// TIA Portal V20 export
FUNCTION_BLOCK "1500Diag82"   // FB82, SCL
{ S7_Optimized_Access := 'TRUE' }
VERSION : 1.1
// stored: MemoryReserve 100, SetENOAutomatically false
   VAR_INPUT
      fId : HW_IO;   // HW-Id of the component from which interrupts are to be received
   END_VAR
   VAR_OUTPUT
      new : Bool;   // A new interrupt was received.
      status : DWord;   // Function result/error message
      id : HW_IO;   // HW-Id of the component (module) from which an interrupt was received
      len : UInt;   // Length of the received interrupt information
      areaLenError : Bool;   // Area length error
   END_VAR
   VAR_IN_OUT
      diag : "typeDiag";   // diagnostics data
   END_VAR
   VAR
      statTinfo { S7_SetPoint := 'True'} : TI_DiagnosticInterrupt;   // Destination area for OB start and management information
      statAinfo { S7_SetPoint := 'True'} : "typeAiPnOrCentral";   // Destination area for header information and additional interrupt information
      statErrorType : USInt;   // Type of error
      statChannelType : USInt;   // Type of channel
      instRalrm { S7_SetPoint := 'True'} : RALRM;   // Instance of RALRM
   END_VAR
   VAR_TEMP
      tempIndex : SInt;
      tempUsint : USInt;
      tempInfo : SInt;
      tempMax : SInt;
      tempReal : Real;
   END_VAR
BEGIN
   //=============================================================================
   // SIEMENS AG
   // (c)Copyright 2017
   //-----------------------------------------------------------------------------
   // Library:       -
   // Tested with:   CPU 1512C-1 PN FW V2.0
   // Engineering:   TIA Portal V14 Update1
   // Restrictions:  call in Diagnostic Error Interrupt OB 82
   // Requirements:  SIMATIC S7-1500 CPU
   // Functionality: Channel diagnostics (PROFINET IO or central I/O)
   //-----------------------------------------------------------------------------
   // Change log table:
   // Version  Date        Expert in charge                 Changes applied
   // 02.00.00 12.01.2017  SIMATIC Industry Online Support  New function: ModuleDiag
   //                                                       & multiple-channelDiag
   //=============================================================================

   // call RALRM in MODE 2 with given F_ID
   #instRalrm(MODE := 2,
              F_ID := #fId,
              NEW => #new,
              STATUS => #status,
              ID => #id,
              LEN => #len,
              TINFO := #statTinfo,
              AINFO := #statAinfo);

   IF (#id = #fId) // some infos will be read every call of OB82
     AND (#statAinfo.addInfo.formatIdentifier = W#16#8000) THEN // W#16#8000: Channel diagnostics 

     #diag.multiError := #statTinfo.MultiError; // =TRUE, if there is more than one error.
     #diag.slotNumber := #statAinfo.header.slotNumber; // Slot number of the component triggering the interrupt
     #diag.submoduleSlotNumber := #statAinfo.header.submoduleSlotNumber; // Submodule slot number of the component triggering the interrupt 
     #tempReal := UINT_TO_REAL(#statAinfo.header.blockLength - 24) / 6; // calculate numbers of multiple-channelDiag
     #tempMax := REAL_TO_SINT(#tempReal) - 1; // calculate upper limit for FOR loop

     FOR #tempInfo := 0 TO #tempMax DO // FOR loop for multiple-channelDiag
       #tempUsint := SHL(IN := #statAinfo.addInfo.diag[#tempInfo].channelErrorType, N := 3); // calculate Type of error
       #statErrorType := SHR(IN := #tempUsint, N := 6); // 1: Incoming error; 2: Outgoing error

       #statChannelType := SHR(IN := #statAinfo.addInfo.diag[#tempInfo].channelErrorType, N := 5); // calculate Type of channel
       // 1: Input channel; 2: Output channel
       //=============================================================================
         IF (#statErrorType = 1) THEN // 1: Incoming error
         //-----------------------------------------------------------------------------      
         IF (#statChannelType = 1) THEN // 1: Input channel

           IF #statAinfo.addInfo.diag[#tempInfo].channelNumber = -32768 THEN // identify module with module diagnostics only
             #diag.moduleDiagOnly := TRUE;
             "ModuleDiag"(errorCode := #statAinfo.addInfo.diag[#tempInfo].errorCode,
                          value := TRUE,
                          diag := #diag.input.module,
                          errorCounter := #diag.errorCounter);
           ELSE
             #diag.moduleDiagOnly := FALSE;

             IF ((#statAinfo.addInfo.diag[#tempInfo].channelNumber >= 0) AND // check array limits (lower limit)
               (#statAinfo.addInfo.diag[#tempInfo].channelNumber <= #diag.input.channel.chMax)) THEN // check array limits (upper limit)
               #diag.input.channel.ch[#statAinfo.addInfo.diag[#tempInfo].channelNumber].error := TRUE; // Set error
               #diag.input.channel.ch[#statAinfo.addInfo.diag[#tempInfo].channelNumber].errorCode := #statAinfo.addInfo.diag[#tempInfo].errorCode; // copy error code
               #diag.errorCounter := #diag.errorCounter + 1; // increment error counter
               #diag.input.channel.areaLenError := FALSE; // Reset area length error
             ELSE
               #diag.input.channel.areaLenError := TRUE; // Set area length error
             END_IF;
           END_IF;
           //-----------------------------------------------------------------------------   
         ELSIF (#statChannelType = 2) THEN // 2: Output channel

           IF #statAinfo.addInfo.diag[#tempInfo].channelNumber = -32768 THEN // identify module with module diagnostics only
             #diag.moduleDiagOnly := TRUE;
             "ModuleDiag"(errorCode := #statAinfo.addInfo.diag[#tempInfo].errorCode,
                          value := TRUE,
                          diag := #diag.output.module,
                          errorCounter := #diag.errorCounter);
           ELSE
             #diag.moduleDiagOnly := FALSE;

             IF ((#statAinfo.addInfo.diag[#tempInfo].channelNumber >= 0) AND // check array limits (lower limit)
               (#statAinfo.addInfo.diag[#tempInfo].channelNumber <= #diag.output.channel.chMax)) THEN // check array limits (upper limit)
               #diag.output.channel.ch[#statAinfo.addInfo.diag[#tempInfo].channelNumber].error := TRUE; // Set error
               #diag.output.channel.ch[#statAinfo.addInfo.diag[#tempInfo].channelNumber].errorCode := #statAinfo.addInfo.diag[#tempInfo].errorCode; // copy error code
               #diag.errorCounter := #diag.errorCounter + 1; // increment error counter
               #diag.output.channel.areaLenError := FALSE; // Reset area length error
             ELSE
               #diag.output.channel.areaLenError := TRUE; // Set area length error
             END_IF;
           END_IF;
           //-----------------------------------------------------------------------------  
         ELSIF (#statChannelType = 3) THEN // 3: Input/output channel

           IF #statAinfo.addInfo.diag[#tempInfo].channelNumber = -32768 THEN // identify module with module diagnostics only
             #diag.moduleDiagOnly := TRUE;
             "ModuleDiag"(errorCode := #statAinfo.addInfo.diag[#tempInfo].errorCode,
                          value := TRUE,
                          diag := #diag.inOut.module,
                          errorCounter := #diag.errorCounter);
           ELSE
             #diag.moduleDiagOnly := FALSE;

             IF ((#statAinfo.addInfo.diag[#tempInfo].channelNumber >= 0) AND // check array limits (lower limit)
               (#statAinfo.addInfo.diag[#tempInfo].channelNumber <= #diag.inOut.channel.chMax)) THEN // check array limits (upper limit)
               #diag.inOut.channel.ch[#statAinfo.addInfo.diag[#tempInfo].channelNumber].error := TRUE; // Set error
               #diag.inOut.channel.ch[#statAinfo.addInfo.diag[#tempInfo].channelNumber].errorCode := #statAinfo.addInfo.diag[#tempInfo].errorCode; // copy error code
               #diag.errorCounter := #diag.errorCounter + 1; // increment error counter
               #diag.inOut.channel.areaLenError := FALSE; // Reset area length error
             ELSE
               #diag.inOut.channel.areaLenError := TRUE; // Set area length error
             END_IF;
           END_IF;
         END_IF;
         //=============================================================================  
       ELSIF (#statErrorType >= 2) THEN // 2: Outgoing error; 3: Outgoing error, other errors present
         //-----------------------------------------------------------------------------
         IF (#statChannelType = 1) THEN  // 1: Input channel

           IF #statAinfo.addInfo.diag[#tempInfo].channelNumber = -32768 THEN // identify module with module diagnostics only
             #diag.moduleDiagOnly := TRUE;
             "ModuleDiag"(errorCode := #statAinfo.addInfo.diag[#tempInfo].errorCode,
                          value := FALSE,
                          diag := #diag.input.module,
                          errorCounter := #diag.errorCounter);
           ELSE
             #diag.moduleDiagOnly := FALSE;

             IF ((#statAinfo.addInfo.diag[#tempInfo].channelNumber >= 0) AND // check array limits (lower limit)
               (#statAinfo.addInfo.diag[#tempInfo].channelNumber <= #diag.input.channel.chMax)) THEN // check array limits (upper limit)
               IF (#statAinfo.addInfo.diag[#tempInfo].errorCode = #diag.input.channel.ch[#statAinfo.addInfo.diag[#tempInfo].channelNumber].errorCode) THEN
                 #diag.input.channel.ch[#statAinfo.addInfo.diag[#tempInfo].channelNumber].error := FALSE; // Reset error
                 #diag.input.channel.ch[#statAinfo.addInfo.diag[#tempInfo].channelNumber].errorCode := 0; // Reset error code
               END_IF;
               #diag.errorCounter := #diag.errorCounter - 1; // decrement error counter
               #diag.input.channel.areaLenError := FALSE; // Reset area length error
             ELSE
               #diag.input.channel.areaLenError := TRUE; // Set area length error
             END_IF;
           END_IF;
           //-----------------------------------------------------------------------------   
         ELSIF (#statChannelType = 2) THEN // 2: Output channel

           IF #statAinfo.addInfo.diag[#tempInfo].channelNumber = -32768 THEN // identify module with module diagnostics only
             #diag.moduleDiagOnly := TRUE;
             "ModuleDiag"(errorCode := #statAinfo.addInfo.diag[#tempInfo].errorCode,
                          value := FALSE,
                          diag := #diag.output.module,
                          errorCounter := #diag.errorCounter);
           ELSE
             #diag.moduleDiagOnly := FALSE;

             IF ((#statAinfo.addInfo.diag[#tempInfo].channelNumber >= 0) AND // check array limits (lower limit)
               (#statAinfo.addInfo.diag[#tempInfo].channelNumber <= #diag.output.channel.chMax)) THEN // check array limits (upper limit)
               IF (#statAinfo.addInfo.diag[#tempInfo].errorCode = #diag.output.channel.ch[#statAinfo.addInfo.diag[#tempInfo].channelNumber].errorCode) THEN
                 #diag.output.channel.ch[#statAinfo.addInfo.diag[#tempInfo].channelNumber].error := FALSE; // Reset error
                 #diag.output.channel.ch[#statAinfo.addInfo.diag[#tempInfo].channelNumber].errorCode := 0; // Reset error code
               END_IF;
               #diag.errorCounter := #diag.errorCounter - 1; // decrement error counter
               #diag.output.channel.areaLenError := FALSE; // Reset area length error
             ELSE
               #diag.output.channel.areaLenError := TRUE; // Set area length error
             END_IF;
           END_IF;
           //----------------------------------------------------------------------------- 
         ELSIF (#statChannelType = 3) THEN // 3: Input/output channel

           IF #statAinfo.addInfo.diag[#tempInfo].channelNumber = -32768 THEN // identify module with module diagnostics only
             #diag.moduleDiagOnly := TRUE;
             "ModuleDiag"(errorCode := #statAinfo.addInfo.diag[#tempInfo].errorCode,
                          value := FALSE,
                          diag := #diag.inOut.module,
                          errorCounter := #diag.errorCounter);
           ELSE
             #diag.moduleDiagOnly := FALSE;

             IF ((#statAinfo.addInfo.diag[#tempInfo].channelNumber >= 0) AND // check array limits (lower limit)
               (#statAinfo.addInfo.diag[#tempInfo].channelNumber <= #diag.inOut.channel.chMax)) THEN // check array limits (upper limit)
               IF (#statAinfo.addInfo.diag[#tempInfo].errorCode = #diag.inOut.channel.ch[#statAinfo.addInfo.diag[#tempInfo].channelNumber].errorCode) THEN
                 #diag.inOut.channel.ch[#statAinfo.addInfo.diag[#tempInfo].channelNumber].error := FALSE; // Reset error
                 #diag.inOut.channel.ch[#statAinfo.addInfo.diag[#tempInfo].channelNumber].errorCode := 0; // Reset error code
               END_IF;
               #diag.errorCounter := #diag.errorCounter - 1; // decrement error counter
               #diag.inOut.channel.areaLenError := FALSE; // Reset area length error
             ELSE
               #diag.inOut.channel.areaLenError := TRUE; // Set area length error
             END_IF;
           END_IF;
         END_IF;
         //============================================================================= 
       END_IF;

       IF #statAinfo.addInfo.diag[#tempInfo].channelNumber <> -32768 AND #statTinfo.Channel = 32768 THEN // for ET200S: no error exists

         FOR #tempIndex := 0 TO #diag.input.channel.chMax DO // delete all input errors
           #diag.input.channel.ch[#tempIndex].error := FALSE; // Reset error
           #diag.input.channel.ch[#tempIndex].errorCode := 0; // Reset error code
         END_FOR;

         FOR #tempIndex := 0 TO #diag.output.channel.chMax DO // delete all output errors
           #diag.output.channel.ch[#tempIndex].error := FALSE; // Reset error
           #diag.output.channel.ch[#tempIndex].errorCode := 0; // Reset error code
         END_FOR;

         FOR #tempIndex := 0 TO #diag.inOut.channel.chMax DO // delete all in-/output errors
           #diag.inOut.channel.ch[#tempIndex].error := FALSE; // Reset error
           #diag.inOut.channel.ch[#tempIndex].errorCode := 0; // Reset error code
         END_FOR;

         #diag.errorCounter := 0; // reset error counter

       END_IF;
     END_FOR;

     IF #diag.errorCounter > 0 THEN // check error counter
       #diag.error := TRUE; // Set module error
     ELSE
       #diag.error := FALSE; // Reset module error
     END_IF;

     IF (#diag.input.channel.areaLenError = TRUE)
       OR (#diag.output.channel.areaLenError = TRUE)
       OR (#diag.inOut.channel.areaLenError = TRUE) THEN
       #areaLenError := TRUE; // set area length error
     ELSIF (#diag.input.channel.areaLenError = FALSE)
       AND (#diag.output.channel.areaLenError = FALSE)
       AND (#diag.inOut.channel.areaLenError = FALSE) THEN
       #areaLenError := FALSE; // reset area length error
     END_IF;

   END_IF;
END_FUNCTION_BLOCK
